FUNCTION_BLOCK Ampel
VAR_INPUT
	e_state_ample : E_STATE_AMPEL;
END_VAR
VAR_OUTPUT
	red:BOOL;
	yellow:BOOL;
	green:BOOL;
END_VAR
VAR
END_VAR

CASE e_state_ample OF
	
	E_STATE_AMPEL.OFF:
		red:=FALSE;
		green:=FALSE;
		yellow:=FALSE;
		
	E_STATE_AMPEL.ALL:
		red:=TRUE;
		green:=TRUE;
		yellow:=TRUE;
	
	E_STATE_AMPEL.RED:
		red:=TRUE;
		green:=FALSE;
		yellow:=FALSE;
		
	E_STATE_AMPEL.YELLOW:
		red:=FALSE;
		green:=FALSE;
		yellow:=TRUE;
		
	E_STATE_AMPEL.GREEN:
		red:=FALSE;
		green:=TRUE;
		yellow:=FALSE;
			
		
END_CASE

END_FUNCTION_BLOCK

(* stored: Version 1.1.0.1, ProductVersion 3.1.4024.13
   POU Ampel: Id {42e454cd-d42b-4e7f-84ee-334959e9c826}, SpecialFunc None *)
